(* IEC 61131-3 sources: generating_plc_code_with_llms/Code#2/Bard/second run, 21 files *)

(* ---- 14.st ---- *)
// 5.19s
// 2
FUNCTION FC1001 :BOOL
VAR_INPUT
  MEW : REAL;
  SP : REAL;
  HYS : REAL;
END_VAR
VAR_IN_OUT
  OUT : BOOL;
END_VAR
VAR
  P_HYS : REAL;
END_VAR

P_HYS := SP * HYS / 100;

IF MEW > SP + P_HYS THEN
  OUT := TRUE;
ELSIF MEW < SP - P_HYS THEN
  OUT := FALSE;
ELSE
  OUT := OUT;
END_IF;

RETURN OUT;
END_FUNCTION

(* ---- 15.st ---- *)
// 6.0s
// 2
VAR
FUNCTION FC1002 :BOOL
VAR_INPUT
  E_A : BOOL;
  SENSOR : BOOL;
  ZEITW : TIME;
END_VAR
VAR_IN_OUT
  ZEIT : TON;
  P_HU : BOOL;
  P_AL : BOOL;
END_VAR

IF E_A THEN
  P1 := TRUE;
ELSE
  P1 := FALSE;
END_IF;

IF SENSOR THEN
  IF ZEIT > 3 THEN
    ZEIT := 0;
    P_HU := FALSE;
    P_AL := TRUE;
  ELSE
    ZEIT := ZEITW;
  END_IF;
ELSE
  P_HU := FALSE;
  P_AL := FALSE;
END_IF;

RETURN P1;
END_FUNCTION

(* ---- 18.st ---- *)
// 5.83s
// 2
FUNCTION FC1003 : VOID
VAR_INPUT
  IN_R:REAL;
  IN_MAX, IN_MIN:REAL;
  OUT_MAX, OUT_MIN:REAL;
END_VAR
VAR_OUTPUT
  OUT_R:REAL;
  FEH:BOOL;
END_VAR
VAR_TEMP
  DIFF1, DIFF2:REAL;
END_VAR

DIFF1 := IN_MAX - IN_MIN;
DIFF2 := OUT_MAX - OUT_MIN;

IF IN_R < IN_MIN THEN
  FEH := TRUE;
  OUT_R := OUT_MIN;
ELSEIF IN_R > IN_MAX THEN
  FEH := TRUE;
  OUT_R := OUT_MAX;
ELSE
  OUT_R := DIFF2 * (IN_R - IN_MIN) / DIFF1 + OUT_MIN;
  FEH := FALSE;
END_IF;

RETURN;
END_FUNCTION;

(* ---- 19.st ---- *)
// 6.5s
// 2
FUNCTION_BLOCK FB1005
VAR_INPUT
  START:BOOL;
  DICKE:REAL;
  V_MAX, V_MIN:REAL;
END_VAR
VAR_OUTPUT
  D_MAX, D_MIN:REAL;
  P1:BOOL;
END_VAR
VAR
  FO:BOOL;
END_VAR

VAR
  MIN_M: REAL;
  MAX_M: REAL;
END_VAR

IF START = TRUE THEN
  FO := FALSE;
  MIN_M := DICKE;
  MAX_M := DICKE;
ELSIF FO = FALSE THEN
  IF DICKE > MAX_M THEN
    MAX_M := DICKE;
  ELSEIF DICKE < MIN_M THEN
    MIN_M := DICKE;
  END_IF;

  IF MAX_M > V_MAX OR MIN_M < V_MIN THEN
    P1 := TRUE;
  ELSE
    P1 := FALSE;
  END_IF;
END_IF;

D_MAX := MAX_M;
D_MIN := MIN_M;

END_FUNCTION;

(* ---- 20.st ---- *)
// 5.81s
// 2
FUNCTION_BLOCK INTERLOCK
VAR_INPUT
  I1 : BOOL;
  I2 : BOOL;
  TL : TIME;
END_VAR
VAR_OUTPUT
  Q1 : BOOL;
  Q2 : BOOL;
END_VAR
VAR
  T1 : TOF;
  T2 : TOF;
END_VAR

Q1 := FALSE;
Q2 := FALSE;

T1(PT := TL);
T2(PT := TL);

WHILE TRUE DO
  IF I1 = TRUE AND Q2 = FALSE THEN
    Q1 := TRUE;
    T1 := 0;
  ELSIF I2 = TRUE AND Q1 = FALSE THEN
    Q2 := TRUE;
    T2 := 0;
  ELSE
    IF Q1 = TRUE THEN
      IF T1.Q THEN
        Q1 := FALSE;
      END_IF;
    ELSE
      IF T2.Q THEN
        Q2 := FALSE;
      END_IF;
    END_IF;
  END_IF;

  WAIT;
END_WHILE;

END_FUNCTION;

(* ---- 21.st ---- *)
// 13.27s
// 2
FUNCTION_BLOCK BURNER
VAR_INPUT
  IN : BOOL;
  STAGE2 : BOOL;
  OVER_TEMP : BOOL;
  OIL_TEMP : BOOL := TRUE;
  FLAME : BOOL;
  RST : BOOL;
  RST_TIMER : BOOL;
  PRE_HEAT_TIME : TIME := t#5s;
  PRE_VENT_TIME : TIME := t#15s;
  PRE_IGNITE_TIME : TIME := t#15s;
  POST_IGNITE_TIME : TIME := t#25s;
  STAGE2_DELAY : TIME := t#10s;
  SAFETY_TIME : TIME := t#5s;
  LOCKOUT_TIME : TIME := t#10s;
  MULTIPLE_IGNITION : BOOL := TRUE;
  KW1 : REAL;
  KW2 : REAL;
END_VAR
VAR_OUTPUT
  MOTOR : BOOL;
  COIL1 : BOOL;
  COIL2 : BOOL;
  PRE_HEAT : BOOL;
  IGNITE : BOOL;
  FAIL : BOOL;
  KWH : REAL;
  STATUS : BYTE;
END_VAR
VAR_IN_OUT
  RUNTIME1 : UDINT;
  RUNTIME2 : UDINT;
  CYCLES : UDINT;
END_VAR
VAR
  state : INT;
  last : TIME;
  tx : TIME;
  last_change : TIME;
  timer1 : TON;
  timer2 : TON;
  oil_temp_last : BOOL;
  cycles2 : UDINT;
END_VAR

// Initialize state and timers
state := 110;
last := TIME := T_CPU;
last_change := T_CPU;
timer1(PT := LOCKOUT_TIME);
timer2(PT := 0);
cycles2 := 0;

WHILE TRUE DO
  // Check for reset and lockout
  IF RST THEN
    IF timer1.Q THEN
      IF NOT OVER_TEMP THEN
        state := 110;
        timer1 := 0;
      END_IF;
    END_IF;
  ELSEIF NOT RST_TIMER THEN
    timer1 := 0;
  END_IF;

  // Check for overall burner shutdown
  IF OVER_TEMP THEN
    state := 110;
    FAIL := TRUE;
    STATUS := 9;
  ELSE
    FAIL := FALSE;

    // State machine for burner operation
    CASE state OF
      110: // Wait for start signal
        IF IN THEN
          state := 111;
          PRE_HEAT := TRUE;
          last_change := T_CPU;
        END_IF;
      111: // Pre-heating
        IF timer1.Q THEN // Lockout if no start after lockout time
          FAIL := TRUE;
          STATUS := 10;
          state := 110;
        ELSIF OIL_TEMP AND T_DEF(last_change - T_CPU) >= PRE_HEAT_TIME THEN
          state := 112;
          MOTOR := TRUE;
          timer1 := 0;
          last_change := T_CPU;
        END_IF;
      112: // Pre-ventilation
        IF timer1.Q THEN // Failure if pre-ventilation time exceeded
          FAIL := TRUE;
          STATUS := 3;
          state := 110;
        ELSIF T_DEF(last_change - T_CPU) >= PRE_VENT_TIME THEN
          state := 113;
          IGNITE := TRUE;
          timer1 := 0;
          last_change := T_CPU;
        END_IF;
      113: // Ignition and post-ignition
        IF timer1.Q THEN // Failure if safety time passed without flame
          FAIL := TRUE;
          STATUS := 4;
          state := 110;
        ELSIF NOT FLAME THEN // Failure if flame detected during ignition
          FAIL := TRUE;
          STATUS := 2;
          state := 110;
        ELSIF T_DEF(last_change - T_CPU) >= POST_IGNITE_TIME THEN
          IF STAGE2 AND T_DEF(last_change - T_CPU) >= STAGE2_DELAY THEN
            cycles2 := cycles2 + 1;
            coil2 := TRUE;
            RUNTIME2 := RUNTIME2 + T_DEF(
        // 26.16s
        ELSIF NOT FLAME AND MULTIPLE_IGNITION THEN
  // Restart ignition if flame absent and multiple ignition enabled
  state := 112;
  IGNITE := FALSE;
  timer1 := 0;
  last_change := T_CPU;
END_IF;
END_CASE;
  END_IF;

  // Update runtime counters and status
  IF state >= 112 THEN
    RUNTIME1 := RUNTIME1 + T_DEF(T_CPU - last);
  END_IF;
  KWH := KW1 * RUNTIME1 + KW2 * RUNTIME2;
  STATUS := state;

  // Update timers
  timer1(IN := state >= 111);
  timer2(IN := state == 113);

  // Update last measurement time
  last := T_CPU;

  WAIT;
END_WHILE;

END_FUNCTION;

(* ---- 1.st ---- *)
// 4.31s
// 2
VAR
    xAllOn : BOOL;
    xAllOff : BOOL;

    xAlarm1 : BOOL;
    xAlarm2 : BOOL;
END_VAR

IF xAllOn THEN
    xAlarm1 := TRUE;
    xAlarm2 := TRUE;
    xAllOn := FALSE;
ELSIF xAllOff THEN
    xAlarm1 := FALSE;
    xAlarm2 := FALSE;
    xAllOff := FALSE;
ELSE
END_IF;

(* ---- 10.st ---- *)
// 4.66s
// 2
VAR_INPUT
  X : REAL;
END_VAR

Sigmoid(X) := 1 / (1 + EXP(-X));

Write_To_Display("Sigmoid(X):", Sigmoid(X));

(* ---- 11.st ---- *)
// 4.81s
// 2
VAR_INPUT
  x : REAL;
END_VAR

Sign(x) := IF x > 0 THEN 1 ELSE -1;

Write_To_Display("Sign(X):", Sign(x));

(* ---- 12.st ---- *)
// 4.59s
// 2
VAR
  X : REAL;
  Sinh : REAL;
END_VAR

Sinh(X) := EXP(X) - EXP(-X) / 2;

Write_To_Display("Sinh(X):", Sinh(X));

(* ---- 13.st ---- *)
// 6.18s
// 2
VAR CONSTANT
  MAXNUMBERS : UINT := 99;
END_VAR

VAR
  aNumbers : ARRAY[0..MAXNUMBERS] OF INT;
  nCnt : INT;
END_VAR

FOR nCnt := 0 TO MAXNUMBERS DO
  aNumbers[nCnt] := RAND();
END_FOR;

REPEAT
  IF aNumbers[nCnt] = 10 THEN
    EXIT;
  END_IF;

  IF aNumbers[nCnt] = targetNum THEN
    FOUND := TRUE;
    EXIT;
  END_IF;

  nCnt := nCnt + 1;
UNTIL (nCnt = MAXNUMBERS) OR FOUND;

IF FOUND THEN
  Write_To_Display("Number found:", targetNum);
ELSE
  Write_To_Display("Number not found:", targetNum);
END_IF;

(* ---- 16.st ---- *)
// 6.98s
// 2
VAR
  North_green : BOOL := FALSE;
  North_yellow : BOOL := FALSE;
  North_red : BOOL := TRUE;
  East_green : BOOL := TRUE;
  East_yellow : BOOL := FALSE;
  East_red : BOOL := FALSE;
  T1 : TON;
END_VAR

T1(PT := 5000ms);

WHILE TRUE DO
  IF T1.Q THEN
    North_green := FALSE;
    North_red := TRUE;
    East_green := FALSE;
    East_yellow := TRUE;
  ELSE
    North_green := FALSE;
    North_yellow := FALSE;
    North_red := TRUE;
    East_green := TRUE;
    East_yellow := FALSE;
  END_IF;

  IF T1.Q THEN
    T1 := 0;
  ELSE
    IF T1.PT >= 9500ms THEN
      East_green := FALSE;
      East_red := TRUE;
      East_yellow := TRUE;
    ELSEIF T1.PT >= 5500ms THEN
      North_green := FALSE;
      North_red := TRUE;
      East_green := TRUE;
      East_yellow := FALSE;
    END_IF;
  END_IF;

  WAIT;
END_WHILE;

(* ---- 17.st ---- *)
// 6.75s
// 2
VAR
  aiOutside : INT;
  aiHumidity: INT;
  sShowText : STRING[80];
END_VAR

aiOutside := Read_Analog_Input;
aiHumidity := Read_Humidity_Input;

IF aiOutside < 18 THEN
  sShowText := "Cold";
ELSIF aiOutside >= 18 AND aiOutside <= 25 THEN
  IF aiHumidity >= 40 AND aiHumidity <= 75 THEN
    sShowText := "Opt";
  ELSE
    sShowText := "Temp. OK";
  END_IF;
ELSIF aiOutside > 25 THEN
  sShowText := "Hot";
END_IF;

Write_Display(sShowText);

(* ---- 2.st ---- *)
// 4.19s
// 3
VAR_INPUT
  N : INT;
  K : INT;
  i : INT;
END_VAR

VAR
  C_nk : INT := 1;
END_VAR

IF K > N THEN
  C_nk := 0;
ELSE
  i := 0;
  WHILE i <= K - 1 DO
    C_nk := C_nk * (N - i);
    C_nk := C_nk / (i + 1);
    i := i + 1;
  END_WHILE;
END_IF;

(* ---- 3.st ---- *)
// 4.52s
// 2
VAR_INPUT
  X : INT;
END_VAR
VAR
  t1 : DINT;
  t2 : DINT;
  x_tmp : INT := 0;
END_VAR

IF X = 0 THEN
  x_tmp := 0;
ELSIF X = 1 THEN
  x_tmp := 1;
ELSE
  t1 := 0;
  t2 := 1;
  FOR i := 2 TO X DO
    x_tmp := t1 + t2;
    t1 := t2;
    t2 := x_tmp;
  END_FOR;
END_IF;

X := x_tmp;

(* ---- 4.st ---- *)
// 4.93s
// 2
VAR
  aiLevel : INT;
  PercentLevel : UINT;
  doLow : BOOL;
  doOk : BOOL;
  doHigh : BOOL;
  doAlarm : BOOL;
END_VAR

CASE aiLevel
  WHEN 0..500 THEN
    PercentLevel := 0;
    doLow := TRUE;
    doOk := FALSE;
    doHigh := FALSE;
    doAlarm := FALSE;
  WHEN 501..1500 THEN
    PercentLevel := (aiLevel - 500) * 2;
    doLow := FALSE;
    doOk := TRUE;
    doHigh := FALSE;
    doAlarm := FALSE;
  WHEN 1501..32767 THEN
    PercentLevel := (aiLevel - 1500) * 4 + 50;
    doLow := FALSE;
    doOk := FALSE;
    doHigh := TRUE;
    doAlarm := FALSE;
  END_CASE;

IF PercentLevel < 1 THEN
  doAlarm := TRUE;
END_IF;

(* ---- 5.st ---- *)
// 5.94s
// 2
VAR
  Start_Loop : BOOL := FALSE;
  one_hour : TIME := T#1h;
  One_Hour_Timer : TON;
  Gate_Open : BOOL := FALSE;
  Close_Gate_Inst : BOOL := FALSE;
  Sensed_Car : BOOL := FALSE;
  Sensed_Car_Inst : BOOL := FALSE;
  Sensed_App : BOOL := FALSE;
  Mobile_Inst : BOOL := FALSE;
  Auth : STRING;
  my_defined_str : STRING := 'abcd';
END_VAR

One_Hour_Timer(PT := one_hour);

IF Start_Loop THEN
  One_Hour_Timer := 0;
END_IF;

IF One_Hour_Timer = 0 AND Gate_Open THEN
  Close_Gate_Inst := TRUE;
END_IF;

IF Sensed_Car OR Sensed_App THEN
  Sensed_Car_Inst := TRUE;
  Mobile_Inst := TRUE;
  IF Input_Auth := Auth AND Auth = my_defined_str THEN
    Gate_Open := TRUE;
    Close_Gate_Inst := FALSE;
    One_Hour_Timer := 0;
  ELSE
    Gate_Open := FALSE;
  END_IF;
END_IF;

IF Sensed_Car_Inst OR Mobile_Inst THEN
  Sensed_Car_Inst := FALSE;
  Mobile_Inst := FALSE;
  IF Gate_Open THEN
    Close_Gate_Inst := TRUE;
  END_IF;
END_IF;

(* ---- 6.st ---- *)
// 6.96s
// 2
VAR CONSTANT
  WAIT : UINT := 0;
  TOP_POSITION : UINT := 1;
  BOTTOM_POSITION : UINT := 2;
  GETBOX : UINT := 3;
  UNLOAD_POSITION : UINT := 4;
  UNLOAD_BOX : UINT := 5;
END_VAR

VAR
  (*-- digital outputs*)
  doConvTop: BOOL := FALSE;
  doConvBottom: BOOL := FALSE;
  doConvLift: BOOL := FALSE;
  doLiftTop: BOOL := FALSE;
  doLiftBottom: BOOL := FALSE;
  doLiftUnload: BOOL := FALSE;
  (*-- digital inputs*)
  diConvTop: BOOL := FALSE;
  diConvBottom: BOOL := FALSE;
  diLiftTop: BOOL := FALSE;
  diLiftBottom: BOOL := FALSE;
  diLiftUnload: BOOL := FALSE;
  diBoxLift: BOOL := FALSE;
  (*-- status variables*)
  selectLift: UINT := WAIT;
  ConvTopOn: BOOL := TRUE;
  ConvBottomOn: BOOL := TRUE;
END_VAR

Main_Control:
  IF diConvTop THEN
    doConvTop := FALSE;
    selectLift := TOP_POSITION;
  END_IF;

  IF diConvBottom THEN
    doConvBottom := FALSE;
    selectLift := BOTTOM_POSITION;
  END_IF;

  IF selectLift = TOP_POSITION THEN
    doLiftTop := TRUE;
    ConvTopOn := FALSE;
  ELSIF selectLift = BOTTOM_POSITION THEN
    doLiftBottom := TRUE;
    ConvBottomOn := FALSE;
  ELSIF selectLift = GETBOX THEN
    doConvLift := TRUE;
    IF diBoxLift THEN
      doConvLift := FALSE;
      selectLift := UNLOAD_POSITION;
    END_IF;
  ELSIF selectLift = UNLOAD_POSITION THEN
    doLiftUnload := TRUE;
    IF diLiftUnload THEN
      doLiftUnload := FALSE;
      selectLift := WAIT;
      ConveyorTopOn := TRUE;
      ConveyorBottomOn := TRUE;
    END_IF;
  END_IF;
END_MAIN_CONTROL;

(* ---- 7.st ---- *)
// 5.28s
// 2
VAR CONSTANT
  MAX_INDEX: USINT := 4;
END_VAR

VAR
  (*-- array of weights *)
  aWeights : ARRAY[0..MAX_INDEX] OF INT;
  (*-- index counter *)
  iCnt : USINT;
  (*-- sum of weights *)
  sumWeight : DINT;
  (*-- average of weights *)
  avgWeight : INT;
END_VAR

FOR iCnt := 0 TO MAX_INDEX - 1 DO
  aWeights[iCnt] := Read_Analog_Input(iCnt);
  sumWeight := sumWeight + aWeights[iCnt];
END_FOR;

avgWeight := sumWeight / MAX_INDEX;

Write_To_Display("Total Weight:", sumWeight);
Write_To_Display("Average Weight:", avgWeight);

(* ---- 8.st ---- *)
// 10.66s
// 2
VAR_INPUT
  X : REAL;
END_VAR
VAR
  w : REAL;
  i : INT;
  we : REAL;
  w1e : REAL;
  ewx : REAL;
  last : DWORD;
END_VAR

we := 0.0;
w1e := 1.0;
ewx := X;
last := 0;

i := 1;
WHILE ABS(w - w1e) > 0.000001 DO
  w := ewx / we;
  w1e := we;
  we := w + ewx / w;

  IF last = 255 THEN
    i := 0;
  END_IF;
  last := last + 1;
END_WHILE;

w := ewx / w;

Write_To_Display("Lambert W(x):", w);

(* ---- 9.st ---- *)
// 5.28s
// 2
VAR
  YEAR : INT;
  isLeapYear : BOOL;
END_VAR

isLeapYear := FALSE;

IF (YEAR % 4 = 0) AND (YEAR % 100 <> 0) OR (YEAR % 400 = 0) THEN
  isLeapYear := TRUE;
END_IF;

Write_To_Display("Is the year ", YEAR, " a leap year?", isLeapYear);
